TYPE UnitBlockGeneric :
UNION
	base : UnitBase;
	controller : UnitController;
	master : UnitIndexerMaster;
	slave : UnitIndexerSlave;
END_UNION
END_TYPE

(* stored: Version 1.1.0.1, ProductVersion 3.1.4020.12
   DUT UnitBlockGeneric: Id {6aac2efd-9672-4072-a66c-eb694838255f} *)
